RoboDK station: DK.rdk

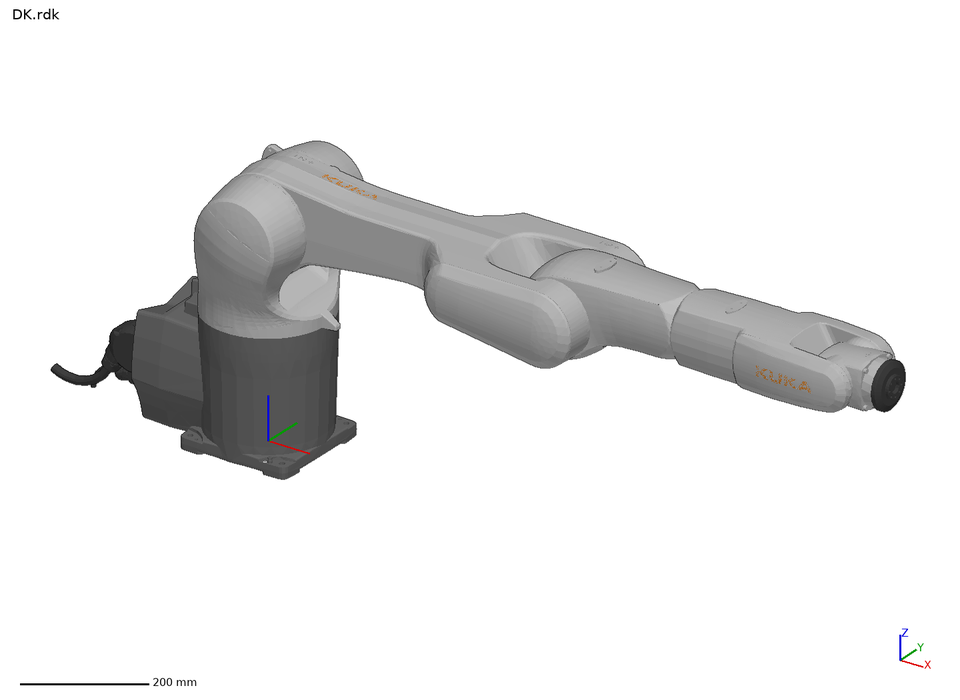
[picture v0: the station drawn from its stored meshes, robots at their saved joint values, targets as dots, program paths as lines]
Station DK (saved by RoboDK 5.9.6). Poses are relative to the parent item; angles as X-Y-Z fixed-axis rotations.
  - frame KUKA KR 10 R1100-2 Base at (0, 0, 0) mm
    - robot KUKA KR 10 R1100-2: 6 axes, payload 10.9 kg, reach 1101 mm, repeatability 0.02 mm, weight 56.5 kg
        modified DH rows (alpha deg, a mm, theta deg, d mm): 0, 0, 0, 400; -90, 25, 0, 0; 0, 560, -90, 0; -90, 25, 0, 515; 90, 0, 0, 0; -90, 0, 180, 90
        joint limits [-170, -190, -120, -185, -120, -350] to [170, 45, 156, 185, 120, 350]; home [0, -90, 90, 0, 0, 0]; saved at [0, 0, 0, 0, 0, 0]
